% RSLogix 500 project Coil Winder.RSS, saved by version 8.30.00.16 %
PROJECT "UNTITLED"    % processor: Bul.1763 MicroLogix 1100 Series B %

PROGRAM FILES
  LAD 2   11 rungs

DATA FILES
  O0 OUTPUT  4 elements
  I1 INPUT  6 elements
  S2 STATUS  66 elements
  B3 BINARY  1 elements
  T4 TIMER  1 elements
  C5 COUNTER  1 elements
  R6 CONTROL  1 elements
  N7 INTEGER  1 elements
  F8 FLOAT  1 elements

LADDER 2
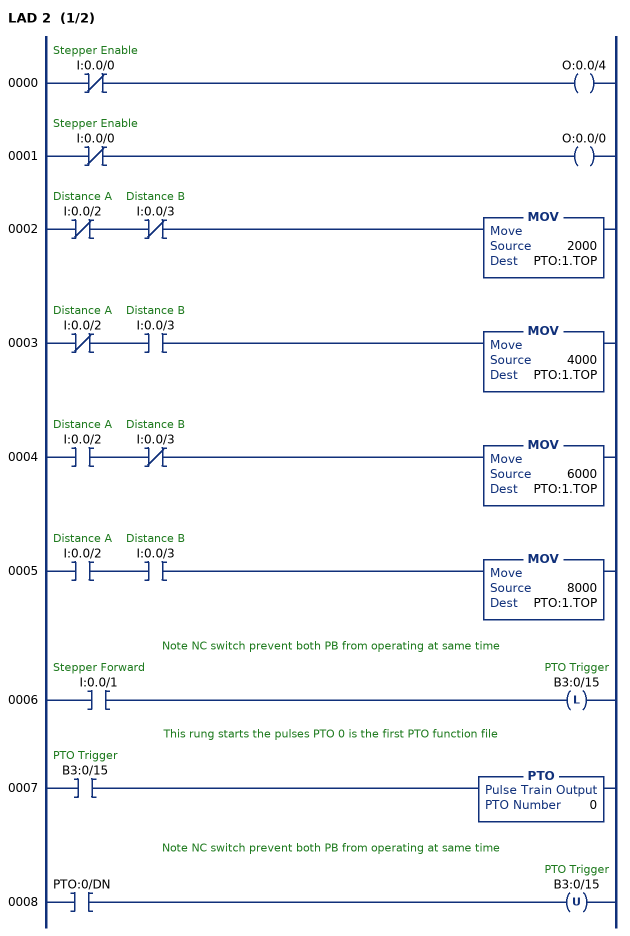
% Rung: 0 %
SOR XIO I:0.0/0 OTE O:0.0/4 EOR
%   I:0.0/0  "Stepper Enable" %
% Rung: 1 %
SOR XIO I:0.0/0 OTE O:0.0/0 EOR
%   I:0.0/0  "Stepper Enable" %
% Rung: 2 %
SOR XIO I:0.0/2 XIO I:0.0/3 MOV 2000 PTO:1.TOP EOR
%   I:0.0/2  "Distance A" %
%   I:0.0/3  "Distance B" %
% Rung: 3 %
SOR XIO I:0.0/2 XIC I:0.0/3 MOV 4000 PTO:1.TOP EOR
%   I:0.0/2  "Distance A" %
%   I:0.0/3  "Distance B" %
% Rung: 4 %
SOR XIC I:0.0/2 XIO I:0.0/3 MOV 6000 PTO:1.TOP EOR
%   I:0.0/2  "Distance A" %
%   I:0.0/3  "Distance B" %
% Rung: 5 %
SOR XIC I:0.0/2 XIC I:0.0/3 MOV 8000 PTO:1.TOP EOR
%   I:0.0/2  "Distance A" %
%   I:0.0/3  "Distance B" %
% Rung: 6 %
% Note NC switch prevent both PB from operating at same time %
SOR XIC I:0.0/1 OTL B3:0/15 EOR
%   I:0.0/1  "Stepper Forward" %
%   B3:0/15  "PTO Trigger" %
% Rung: 7 %
% This rung starts the pulses PTO 0 is the first PTO function file %
SOR XIC B3:0/15 PTO 0 EOR
%   B3:0/15  "PTO Trigger" %
% Rung: 8 %
% Note NC switch prevent both PB from operating at same time %
SOR XIC PTO:0/DN OTU B3:0/15 EOR
%   B3:0/15  "PTO Trigger" %

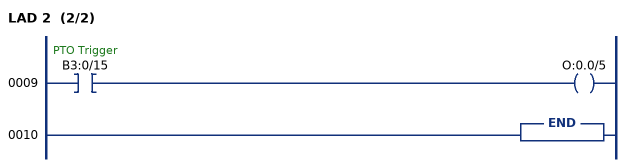
% Rung: 9 %
SOR XIC B3:0/15 OTE O:0.0/5 EOR
%   B3:0/15  "PTO Trigger" %
% Rung: 10 %
SOR END EOR

OTHER DOCUMENTED ADDRESSES
  B3:0/0  "STEP On or Off"
  B3:0/1  "Trigger to change pulse number"
  B3:0/4  "Trigger to change pulse frequency"
  B3:0/7  "Forward Run"
  B3:0/8  "Reverse Run"
  O:0.0/3  "Direction Bit"

COMMENTS NOT ATTACHED TO A CURRENT RUNG
  B3:0/8: Rung for choosing reverse direction
  B3:0/7: Rung for choosing forward direction
  PTO:0.6: This rung if for sending number of pulses to pulse train register for PTO 1
